(* IEC 61131-3 sources: Dev/Dev_V200/200 (part 18) *)

(* ---- _Nh_WEB.st ---- *)
(* KNIZNICA PRE FUNKCIE WEBMAKERU: HomePage,autologin, presmerovanie na volnu stranku a riadenie pristupu = usermanagement, *)

{ $ IFDEF __NH_WEB }

// hlavna obrazovka

// ************************** web ****************

FUNCTION _NhTchObjOK   {HIDDEN} : BOOL                                     // dotyk nad aktivnym objektom ( cm>0) na stranke
	VAR_INPUT
		///***26.6.24 skusmo pridane pre 109
		Qr			: BOOL;						// posle hned v 1.cykle po dotyku aj CMD, cim zabezpeci refresh a prijatie xA^.tch.Qr
		obj		: BOOL := true;
		cmd		: USINT;
	END_VAR
	IF Obj THEN
   	xA^.tch.cm     := xO^.cm;
	ELSE
		xA^.tch.cm     := cmd;
	END_IF;

   xA^.tch.row    := j;                               // tu sa vyplni ak by nebol browser
   xA^.tch.obj    := INT_TO_SINT(ix);
   xA^.tch.Q      := true;                            // centralny priznak, ze na nejakom objekte bol dotyk
   xA^.tch.Qr     := true;
   xO^.tch        := true;                            // priznak dotyku priamo na objekte, nuluje ho xA^.tch.Qf a do objektu uz nedojde
	xA^.tch.aObj	:= PTR_TO_UDINT( ADR(xO^) );
 	xO^.Q				:= true;									// nastavi sa Qr, zostane v objekte aj po Qf, objekt si ho spolu s Qf musi vynulovat sam
	IF Qr	THEN
		xA^.tch.CMD    := xA^.tch.cm;							// refresh v tom cykle je este xA^.tch.Qr := true
   	xO^.Qr			:= true;                         // cita sa v objekte, nuluje sa v dalsom cykle
	END_IF;
   ix             := 0;                                              // vykona sa exit s WHILE
   j              := 0;
   _NhTchObjOK       := true;

 	_Nh_Log_Evn_ADD(tsk := 200);

END_FUNCTION

FUNCTION _NhObjXY {HIDDEN}: BOOL                                     // dotyk nad aktivnym objektom ( cm>0) na stranke
   _NhObjXY := false;
   IF xA^.tch.x1 > xO^.x - x  AND
      xA^.tch.x1 < xO^.x + x  AND
      xA^.tch.y1 > xO^.y - y  AND
      xA^.tch.y1 < xO^.y + y  THEN

      _NhTchObjOK();
      _NhObjXY       := true;
   END_IF;
END_FUNCTION

FUNCTION _NhTchObj  {HIDDEN} : BOOL            // zaciatok noveho dotyky = hlada sa objekt
   VAR_TEMP
		wh2r		: BOOL;
      o        : INT;
      wh       : USINT;
//      whOld    : USINT;
	END_VAR
   _NhTchObj      := false;
   j  := USINT_TO_SINT(xM^.ixb[0].row.rws);
   WHILE _NhTchObj = false AND j > 0 AND xA^.tch.row < 0 DO
      IF xB^.r[ j ].h.nd > 0  THEN                                	// j = riadok
         xR    := ADR(xB^.r[ j ]);
         ix  	:= SINT_TO_INT(_RowObr);                              // ix = objekt; max.pocet objektov
         WHILE _NhTchObj = false AND  ix >= 0 DO                     // posupuje sa od posledneho objektu (je navrchu ) az k 0-temu, ktory je naspodku (oramovanie browsu)
				wh2r 	:=	false;
				IF ix > 0 THEN
            	xO    :=  ADR(xR^.o.ob[ix-1]);                           // predchadzajuci riadok
      			wh2r 	:= xO^.wh=123 OR  xO^.wh=109;							// preskoci aktualny riadok
				END_IF;
   			xO    :=  ADR(xR^.o.ob[ix]);
            IF wh2r 	 THEN
					;
            ELSIF xO^.nTch OR xO^.wh =  0 THEN
					;
            ELSIF xO^.wh = 13 THEN
            	o        		:= xO^.fn;
             	xS       		:= ADR(xB^.s[o]);
					IF xB^.s[xO^.fn].zom AND
						_NhTchObjXYW(	x	:=	xO^.x + xO^.w - 100,
											y 	:= xO^.y-50,
											w 	:= 100,
											h	:= 30 		 )	THEN

						xB^.s[xO^.fn].tun := NOT xB^.s[xO^.fn].tun;        // zmeni tun/sld/tun...
                  _NhTchObj      := _NhTchObjOK();
                  xO^.tch   		:= false;                                           // nastavi sa okamzite dotyk
                  xA^.tch.cmd    := xA^.tch.cm;                                           // nastavi sa okamzite dotyk
						xA^.tch.end		:= true;

         		ELSIF _NhTchObjXYW(	x	:=	xO^.x-15,
												y 	:= xO^.y-10,
												w 	:= xO^.w+30,
												h	:= 20 		 ) THEN

							IF (  xS^.bal AND xA^.tch.x1 > xS^.xv - 15 AND xA^.tch.x1 < xS^.xv + 15 ) // je zobrazena gulicka, dotyk na nej okamzite vyvola slider
                              OR
                           (  xA^.tch.x1 > xO^.x - 15 AND xA^.tch.x1 < xO^.x + 15)                // alebo dotyk okolo zaciatku
                              OR
                              xL^.brw = false   THEN

	                        _NhTchObj      := _NhTchObjOK();
  	                        xA^.tch.cmd    := xA^.tch.cm;                                           // nastavi sa okamzite dotyk
									xA^.tch.evn 	:= 6;

                     END_IF;
					END_IF;

            ELSIF xO^.wh = 14 THEN      // point-time SLIDER
            	IF xA^.tch.y1 > xO^.y - xO^.h AND                        // pod vrchom
                        xA^.tch.y1 < xO^.y + 50   AND                         // pod spodkom = obrazok
                        xA^.tch.x1 > xO^.x - 60    AND                        // pred zaciatkom
                        xA^.tch.x1 < xO^.x + xO^.w + 60    THEN               // za koncom
                        _NhTchObj      := _NhTchObjOK();

								xA^.tch.evn 	:= 6;
                        xA^.tch.cmd    := xA^.tch.cm;

						END_IF;

            ELSIF xO^.wh = 123 THEN      // vyber z volieb {riadkov} pod sebou  - NOVA VERZIA
               // tento objekt je dvojriadkovy, v druhom riadku sa vyhodnocuje WhOld z predch.riadka
               xOh := xO;
               IF xA^.tch.x1 >= xOh^.cf.x - 10                             AND     // 1.riadok zaciatok
                  xA^.tch.x1 <= xOh^.cf.x + xOh^.cf.w                         AND     // 1.riadok koniec
                  xA^.tch.y1 >= xOh^.cf.y - 20                             AND     // 1.riadok zaciatok
                  xA^.tch.y1 <= xOh^.cf.y + USINT_TO_INT(xOh^.cf.rw2)*xOh^.cf.h  THEN    // posledny riadok  (+10 je akokeby riadok naviac)

						_NhTchObj      := _NhTchObjOK(obj:=false,cmd:=205);
//                  xA^.tch.cm     := 251;
//                  xA^.tch.cm     := 205;
                  xOh^.tch       := true;                                           // priznak dotyku priamo na objekte

               END_IF;
//            ELSIF WhOld = 123 THEN       // prepinac medzi riadkami - NOVA VERZIA
               ;
            ELSIF xO^.wh = 103 THEN      // vyber z volieb {riadkov} pod sebou  - NOVA VERZIA
               ;
            ELSIF xO^.wh = 107 THEN      //  doplnujuce statusy na objektom
               IF _Nh_Web_SHW_107(tch:=true) THEN
                  _NhTchObj      := true;
               END_IF;
            ELSIF xO^.wh = 109 THEN      //  ROL * slider
            	xRo				:= xO;
               IF _NhxPt(c := xRo^.cf.c, n := xRo^.cf.n,x:=109) = false THEN
               	RETURN;
					END_IF;
               xRol 				:= xPt;
					xRol^.me.CMDs	:= 0;																		// reset
(*
					IF _NhxCfg(c := xRo^.cf.c, n := xRo^.cf.n, par := true, p := xRo^.cf.p, x:=20) = false THEN
						RETURN;
					END_IF;
*)

					del := USINT_TO_INT(xRo^.wObr);											// len prevod na INT - koli strukture

					IF xRo^.StatRow AND
						_NhTchObjXYW(		x := xRo^.xObrL - del/2 ,        				// dotyk nad ikonou LAM v stavovom riadku
												y := xRo^.yObr  - del/2 ,
												w := del,
												h := del) THEN
							_NhTchObj      := _NhTchObjOK( Qr:=true );
							xRol^.me.CMDs	:= 28;													// Lamely do opacneho smeru

					ELSIF xRo^.StatRow AND
							_NhTchObjXYW(	x := xRo^.xObrR - del/2 ,        				// dotyk nad ikonou ROL v stavovom riadku
												y := xRo^.yObr  - del/2 ,
												w := del,
												h := del) THEN
							_NhTchObj      := _NhTchObjOK( Qr:=true );
							xRol^.me.CMDs	:= 11;													// ROLETA prepnut

//					ELSIF xRol^.cx.etHandBlkWind > 0 AND														// bezi delay rucneho zasahu
					ELSIF xRol^.cx.CmdWind = 20 AND														// bezi delay rucneho zasahu
							_NhTchObjXYW(	x := xRo^.x + xRo^.w - xRo^.wObrInfo/2,		// zrusit delay rucneho zasahu
												y := xRo^.y - xRo^.wObrInfo/2,
												w := xRo^.wObrInfo,
												h := xRo^.wObrInfo) THEN
							_NhTchObj      := _NhTchObjOK( Qr:=true );
							xRol^.me.CMDs	:= 200;													// zrusit blokovanie

					ELSIF xRol^.cx.CmdWind = 10 AND												// bezi ochrana pred vetrom - restartnut
							_NhTchObjXYW(	x := xRo^.x - xRo^.wObrInfo/2,
												y := xRo^.y - xRo^.wObrInfo/2,
												w := xRo^.wObrInfo,
												h := xRo^.wObrInfo) THEN
							_NhTchObj      := _NhTchObjOK( Qr:=true );
							xRol^.me.CMDs	:= 201;													// restart WindGuard

					ELSIF xRo^.SldLam AND xRo^.tchLam AND										// slider LAM
							_NhTchObjXYW(	x := xRo^.xLam - 10 ,
												y := xRo^.yLam - xRo^.rCirSld/2,
												w := 20,
												h := xRo^.hLam + xRo^.rCirSld) THEN
							_NhTchObj      := _NhTchObjOK( Qr:=true );
							xA^.tch.evn 	:= 6;
							xRol^.me.CMDs	:= 72;													// slider LAM

    				ELSIF _NhTchObjXYW(	x := xRo^.x  ,											// plocha rolety aj s boxom nad
												y := xRo^.y - xRo^.bRol,
												w := xRo^.w ,
												h := xRo^.h + xRo^.bRol + xRo^.rCirSld ) THEN

							_NhTchObj      := _NhTchObjOK( Qr:=true );
							IF xRo^.SldRol THEN                                         // povoleny slider
								xA^.tch.evn 	:= 6;
								xRol^.me.CMDs	:= 71;												  	// slider ROL
							ELSIF xRo^.tchUpDn  THEN                             			// povolit prepnutie
								xRol^.me.CMDs	:= 1;														// prepni
							ELSE
								xRol^.me.CMDs	:= 3;														// stop
							END_IF;
					END_IF;
					IF _NhTchObj AND xRo^.chk = false AND xRol^.cx.CMD > 200 THEN
						xA^.tch.evn 	:= 0;
						xRol^.me.CMDs	:= 3;													// restart WindGuard
      			END_IF

            ELSIF xO^.wh = 22 OR xO^.wh = 121 THEN      														//  HET/VEN : AUTO-MAN/0/1/2/3
//					IF _NhTchObjXYW(x:=xO^.x-xO^.w/2, y:=xO^.y-xO^.w/2, w:=xO^.h * 4 + xO^.w, h := xO^.w) THEN
					IF _NhTchObjXYW(x:=xO^.x-xO^.w/2, y:=xO^.y-xO^.w/2, w:=xO^.h * USINT_TO_INT(xO^.cf.c) + xO^.w, h := xO^.w) THEN
						_NhTchObj      := _NhTchObjOK();
					END_IF;

            ELSIF xO^.wh = 21  THEN
					IF _NhTchObjXYW(x:=xO^.x-xO^.w/2, y:=xO^.y-xO^.w/2, w:=xO^.w, h := xO^.w) THEN
						_NhTchObj      := _NhTchObjOK();
					END_IF;

            ELSIF xO^.wh > 0 AND xO^.nTch = false THEN

               x     := xO^.w / 2 + 9;
               y     := x;             //***

               // xO^.h : 1 - obrazok s  podfarbenim
               // 6 - vypis textu :vyska
               // 10 - obrazok WSB
               // 13 - slider
               // 16 - bool premenna
               // 17 - akcie na obrazovke k WSB
               // 19 - vypisanie hodnoty premennej : style
               // 20 - chceck nad polom obrazkov
               // 21 - vypis textu s hodnotou
               // 90 - dash h=vyska       OK
               CASE xO^.wh OF
//                 22 :   wh := 20;
                120 :   wh := 255;
               ELSE     wh := xO^.wh;
               END_CASE;

               CASE wh OF
                  0 : ;                                              // prazdny objekt
                255 :   // objekt je urceny sirkou a vyskou, vo vnutri moze mat podobejky, ktore sa identifikuju v _Nh_SHW
                        IF xA^.tch.x1 >= xO^.x - xO^.h/2          AND      // spodna hranica = zaciatok - vyska/2
                           xA^.tch.x1 <= xO^.x + xO^.w + xO^.h    AND      // horna hranica
                           xA^.tch.y1 >= xO^.y - xO^.h/2          AND      // vrch
                           xA^.tch.y1 <= xO^.y + xO^.h/2  THEN             // spodok
                           _NhTchObj := _NhTchObjOK();
                        END_IF;

                  6 :   // click nad textom formatovany je zlava do prava
                     ok := xA^.tch.y1 > xO^.y - 20 AND xA^.tch.y1 < xO^.y + 20;
                     CASE xO^.fn  OF
                       2 : // na stred
                           ok := ok AND xA^.tch.x1 > xO^.x - xO^.w/2 AND xA^.tch.x1 < xO^.x + xO^.w/2;
                       1 : // z prava do lava
                           ok := ok AND xA^.tch.x1 > xO^.x - xO^.w AND xA^.tch.x1 < xO^.x;

                     ELSE  // zlaba do prava
                           ok := ok AND xA^.tch.x1 > xO^.x AND xA^.tch.x1 < xO^.x + xO^.w;

(*
                        IF xA^.tch.x1 > xO^.x           AND
                           xA^.tch.x1 < xO^.x + xO^.w   AND
                           xA^.tch.y1 > xO^.y - 20   AND
                           xA^.tch.y1 < xO^.y + 20 THEN
                           _NhTchObj      := _NhTchObjOK();
                        END_IF;
*)
                     END_CASE;
                     If ok THEN
                        _NhTchObj      := _NhTchObjOK();
                     END_If;

                 15 : // typovy DAY + PO-NE
                        xPtD  := ADR(xO^.cf.n);                                                             // na adrese xO^.cf.n + xO^.cf.p je adresa premennej v UDINT
                        xPoD  := UDINT_TO_PTR(xPtD^);

                        _Nh_FRM_Read(frm:=248);   // sablona PO-NE pre DAY,HET,VEN
                                                                       // pointer riadiacej jstruktury dna
                        xM^.pod.po.Btn := false;
                        IF    xA^.tch.y1 > xO^.y - 40 AND                                    // vrchny okraj typovyc dni
                              xA^.tch.y1 < xO^.y + 85+35 THEN                                // spodny okraj PO-NE
                           // sme v objekte
                           FOR i := 0 TO 11 DO
                              IF i > 0 AND i < 8 THEN
                                 y := xO^.y + 85;                                         // dni Pon-Ned
                              ELSE
                                 y := xO^.y;
                              END_IF;
                              IF xA^.tch.y1 < y + 40 AND                                  // nad spodkom
                                 xA^.tch.y1 > y - 40 AND                                  // pod vrchom
//                                 xA^.tch.x1 < xO^.x + _ObjDay.xDay[i]+40 THEN             // pred koncom objektu
                                 xA^.tch.x1 < xO^.x + yFrm_248.xDay[i]+40 THEN             // pred koncom objektu

                                 xM^.pod.po.Btn := xM^.pod.po.Day = i;                            // stlaceny ten isty BTN
                                 IF xM^.pod.cp.cpy THEN                                       // je oznacene kopirovanie
                                    IF xM^.pod.po.Btn = false THEN                            // vymazat vsetko ku kopirovaniu
                                       xM^.pod.cp.dst[i] := NOT xM^.pod.cp.dst[i];
                                    END_IF;
                                 ELSIF i = 0 THEN                                         // prepli sme na hlavmu ikonu prac.dni
                                    IF xPoD^.Day=0 OR xPoD^.Day > 7 THEN                  // predtym bola ina hlavna ikona
                                       xPoD^.Day := _Nh_Poi_Home_Day();                        // nastavi sa aktualny day
                                    END_IF;
                                    xM^.pod.po.Day := xPoD^.Day;
                                 ELSE

                                    IF xPoD^.Day = 0 THEN
                                       xPoD^.Day := i;                                    // prepnutie na iny den a ked je fix prepise Day
                                    END_IF;
                                    xM^.pod.po.Day := i;
                                 END_IF;
                                 _NhTchObj   := _NhTchObjOK();
                                 EXIT;
                              END_IF;
                           END_FOR;
                        END_IF;

                 10 : // akcie od WSB, typ spotrebica (v xO^.h je cislo obrazka)
                     _NhTchObj   := _NhObjXY();

                 17 : // akcie od WSB, typ spotrebica (v xO^.h je cislo obrazka)
                     _NhTchObj   := _NhObjXY();
                 19 : // text
(*
                  GTEXT_STYLE_ITALIC + GTEXT_STYLE_ALIGN_LEFT   + GTEXT_STYLE_HRIGHT  + GTEXT_STYLE_VCENTER,    // stred riadka zlava do prava
                  GTEXT_STYLE_ITALIC + GTEXT_STYLE_ALIGN_RIGHT  + GTEXT_STYLE_HLEFT   + GTEXT_STYLE_VCENTER,    // stred riadka, zprava do lava
                  GTEXT_STYLE_ITALIC + GTEXT_STYLE_ALIGN_CENTER + GTEXT_STYLE_HCENTER + GTEXT_STYLE_VCENTER,    // stred riadka, stred textu
                  GTEXT_STYLE_NORMAL + GTEXT_STYLE_ALIGN_LEFT   + GTEXT_STYLE_HRIGHT  + GTEXT_STYLE_VDOWN,       // zhora-dolu, zlava do prava
                  GTEXT_STYLE_NORMAL + GTEXT_STYLE_ALIGN_RIGHT  + GTEXT_STYLE_HRIGHT  + GTEXT_STYLE_VDOWN       // zhora-dolu, zlava do prava
*)
                     IF xO^.fn = 0 THEN
//                        y := xO^.h/2+5;
                        y := xO^.h*2  ;
                        CASE xO^.BgC OF
                          0 : x := -xO^.w/2;
                          1 : x := xO^.w/2;
                          3 : ;
                          4 : ;
                        END_CASE;
                        IF xA^.tch.y1 > xO^.y - y AND                        // pod vrchom
                           xA^.tch.y1 < xO^.y + y   AND                         // pod spodkom = obrazok
                           xA^.tch.x1+x > xO^.x - xO^.w/2    AND                        // pred zaciatkom
                           xA^.tch.x1+x < xO^.x + xO^.w/2    THEN               // za koncom
                           _NhTchObj      := _NhTchObjOK();
                        END_IF;
                     ELSE
                        _NhTchObj := _NhObjXY();
                     END_IF;

                 27 : // viac BOOL premennych v poli za sebou (DayMode+LOCK)
                        IF _NhObjXY() THEN
                           xO^.tch := 1;
                           _NhTchObj := true;
                        END_IF;

                 20 : // viac BOOL premennych v poli za sebou (DayMode+LOCK)
                     IF xO^.cf.c > 0 AND xO^.h = 0 THEN  // viac objektov na sebe, cislo objektu je ulozene v premennej, ktora je USINT, prepne na dalsi objekt
                        IF _NhObjXY() THEN
                           _NhTchObj := true;
                           xPtD  := ADR(xO^.cf.n);                                                             // na adrese xO^.cf.n + xO^.cf.p je adresa premennej v UDINT
                           xPtU  := UDINT_TO_PTR(xPtD^);
                           IF xPtU^ < xO^.cf.c THEN
                              xPtU^ := xPtU^ + 1;
                           ELSE
                              xPtU^ := 0;
                           END_IF;
                        END_IF;
                     ELSE
                        x := xO^.w/5*3;
                        IF xA^.tch.x1 > xO^.x - x  AND                            // tesne pred prvym obrazkom
                           xA^.tch.x1 < xO^.x + x + xO^.h * USINT_TO_INT(xO^.cf.c)  AND       // tesne za poslednym obrazkom
                           xA^.tch.y1 > xO^.y - x  AND
                           xA^.tch.y1 < xO^.y + x  THEN
                           _NhTchObj      := _NhTchObjOK();
                        END_IF;
                     END_IF;

                 23 :   // prepinac viac riadkov pod sebou
                        y := USINT_TO_INT(xO^.cf.c);
                        IF xA^.tch.x1 > xO^.x - 10          AND     // zaciatok komponenty
                           xA^.tch.x1 < xO^.x + xO^.w + 10  AND     // koniec
                           xA^.tch.y1 > xO^.y - 20          AND     // 1.riadok
                           xA^.tch.y1 < xO^.y + (xO^.fn * y) + 20   // posledny riadok
                                 THEN
                           _NhTchObj   := _NhTchObjOK();
                           o           := xO^.y + xO^.fn/2;
                           FOR i := 1  TO xO^.cf.c DO
                              IF xA^.tch.y1 < o THEN
                                 xFmt23      := ADR(xO^.fmt);
                                 xFmt23^.obj := i;
//                                 xA^.tch.prs := false;
                                 EXIT;
                              END_IF;
                              o := o + xO^.fn;
                           END_FOR;
                        END_IF;

//                 21 :   // prepinac viac riadkov pod sebou
//   	                  y     := x;
//	   	               _NhTchObj := _NhObjXY();

               ELSE
                  IF xO^.h <= 0 THEN
                     y     := x;
                  ELSE
                     y     := xO^.h / 2 + 9;
                  END_IF;
                  _NhTchObj := _NhObjXY();
               END_CASE;
            END_IF;
            IF _NhTchObj THEN
               RETURN;
            END_IF;
            ix       := ix - 1;
//            ix       := ix + 1;
//            WhOld    := xO^.wh;                 // pre dvojriadkove objekty (123..)

         END_WHILE;
      END_IF;
      j := j - 1;
   END_WHILE;
END_FUNCTION

FUNCTION _NhTchMnu {HIDDEN} : BOOL      // najde riadok a v nom objekt na ktorom bol dotyk
  _NhTchMnu       := false;

  xA^.tch  := _eTch;
  aWht     := _eWht;

   xA^.tch.x1     := xCan^.touch.x;
   xA^.tch.x2     := xCan^.touch.x ;
   xA^.tch.y1     := xCan^.touch.y;
   xA^.tch.y2     := xCan^.touch.y;

   jj    := 8;                                                 // prechadzaju sa vsetky menu
   rb    := false;
   IF xM^.edt  THEN
      jj := 1;                                                                // testuje sa len CANCEL
   ELSIF xB^.rw > 0 AND xL^.brw THEN                                          // ak je browser a su naplnene nejake riadny, najskor pg navigator
      IF _NhTchXY(v := xA^.tch.y1, v1 := ky2, v2 := ky2, xy:= 30 ) THEN         // dotyk okolo  spodnej ciary
         x := xIxB^.x1;
         FOR i := 1  TO xIxB^.n DO
            IF _NhTchXY(v := xA^.tch.x1, v1 := x, v2 := x, xy := 30 ) THEN     // dotyk nad bodom
               IF xIxB^.idx > xIxB^.row.rws THEN                               // mame viac dat zaznamov ako je riadkov
                  IF i = xIxB^.n THEN                                          // posledny index
                     i := xIxB^.idx - xIxB^.row.rws + 1;
                  ELSIF i = 1 THEN                                             // 1.index
                     ;
                  ELSE
                     i := (i-1) * xIxB^.row.rws  + 1;                          // vypocita sa
                  END_IF;
               ELSE
                  i := 1;
               END_IF;
               _Nh_Map_Idx(ixb := 0, idx := i);                                  // namapuje najdeny index
               xIxB^.ix1   := i;                                               // toto asi nemusi byt
               xL^.rw1     := xIdx^.ix[aWeb.nbr].dev;                              // do 1.riadku sa vlozia data
               xA^.tch.cmd := 252;                                             // vypis a predefinovanie dat od noveho 1-veho riadka
               _NhTchMnu   := true;
               RETURN;
            END_IF;
            x := x + USINT_TO_INT(xIxB^.w);
         END_FOR;

			// dotyk na spodnej ciare mimo PG-navigator tu sa meni mierka yk:=1.0 .... yk       := MIN(xUsr^.cx.IP[1].y, 1.14) ;

		END_IF;
      ;
   END_IF;
   FOR j := 1  TO jj DO
      xOm  := ADR(xU^.o[j]);
      IF xOm^.fn > 0 AND  xOm^.cm > 0 AND
         _NhTchXY(v := xA^.tch.x1, v1 := xOm^.x, v2 := xOm^.x, xy:= xOm^.w/7*4 )  AND // sirka
         _NhTchXY(v := xA^.tch.y1, v1 := xOm^.y, v2 := xOm^.y, xy:= xOm^.w/7*4 )    // vyska
            THEN
         xA^.tch.obj  := j;
         xA^.tch.cm   := xOm^.cm;
         IF xL^.obj = 200 AND xA^.tch.obj > 2 THEN              // stlacene spodne menu v SETUP
            xA^.tch.cmd    := 200;
         ELSE
            xA^.tch.cmd  := xA^.tch.cm;
         END_IF;
         _NhTchMnu    := true;
         EXIT;
      END_IF;
   END_FOR;
   IF xM^.edt  THEN                                            // edituje sa nazov
      IF _NhTchMnu THEN
         xM^.new := -1;
      END_IF;
       xA^.tch.cmd      := 100;                                // aktivuje CMD editaciu okamzite
      _NhTchMnu         := true;
   ELSIF xA^.tch.x1 > xc - 150         AND                     // dotyk na nazve
         xA^.tch.x1 < xc + 150         AND
         xA^.tch.y1 > xU^.o[1].y - 20  AND                     // vyska nazvu
         xA^.tch.y1 < xU^.o[1].y + 20 THEN

      IF xF^.cf.c = 0 OR xF^.cf.n = 0 THEN                     // nazvy su z aLang
            ;
      ELSIF xM^.set THEN
         rb := aCfg[xL^.fil.cf.c].edn;                         // cfg, vratane nazvy Moj domov co je acfg[3] = zone
      END_IF;
      IF rb THEN
//			xA^.trg.Qr     := 0;
//			xA^.trg.Qf     := 0;
//			xA^.trg.Q      := 0;
         xA^.tch.cmd    := 101;                                // aktivuje CMD editaciu okamzite
         xM^.edt        := true;                               // pri modifikacii nazvu sa to oznaci hned
         _NhTchMnu      := true;
      END_IF;
   END_IF;
END_FUNCTION

FUNCTION_BLOCK _NhWebAcces   {HIDDEN}
   VAR_TEMP
      s        : USINT;
      sa       : USINT;
//      new      : STRING[14];
   END_VAR
   GetWebServerAccess(accessTable := aAcc.wA);
   IF aAcc.wA <> aAcc.wO OR SYSTEM_S.F_EDGE_1SEC THEN
      aAcc.WebChg := aAcc.WebChg + 1;                                         // pocet zmien
      memset(0, sizeof(aAcc.pgN), void(aAcc.pgN));                          // vymazat novy pg, ktorasa bude naplnat
      ii := aWeb.A[1].usr;
      FOR aWeb.nbr := 1 TO _Nh_WEB_M DO
         aWeb.A[ aWeb.nbr ].usr := 0;
      END_FOR;
      FOR s := 0 TO 7 DO
         sa    := _webState(s := aAcc.wA[s].state);
         IF sa = 3  THEN                                                      // zaujima nas len stav 3
            yTx3  := MID(aAcc.wA[s].lastFile,8,5);                            // "/002_NHM.XML" .... '_NHM.XML'
            IF yTx3 = '_NHM.XML' THEN                                           // nova stranka je Mx                           OK
               yTx3  := MID(aAcc.wA[s].lastFile,3,2);
               i := STRING_TO_USINT(yTx3);
               IF i <= _Nh_WEB_M THEN
                  aWeb.A[ i ].usr := i;
                  IF aWeb.M[ i ].naz = '' AND  aWeb.M[ i ].new < 1 THEN
                     aWeb.A[ i ].tch.cmd := 20;                   // vytvori sa nova obrazovka
                     aWeb.M[ i ].lvl     := 0;
                  END_IF;
               END_IF;
            END_IF;
         END_IF;
      END_FOR;
      IF aWeb.A[1].usr > 0 AND ii > 0 THEN
//         aWeb.A[1].usr := ii;
      END_IF;
      aAcc.wO  := aAcc.wA;                                            // vyrovna data
   END_IF;
END_FUNCTION_BLOCK

FUNCTION_BLOCK _NhWebControl    {HIDDEN}
  	VAR
      fbNhWebAcces : _NhWebAcces;
  	END_VAR
      fbNhWebAcces();                                                // riadenie pristupu na webserver
      // prechadza nadefinovane stranky
      FOR aWeb.nbr := 1 TO _Nh_WEB_M DO
//         IF aAcc.pgN.pg[aWeb.nbr].usage > 0 THEN                   // aktivna stranka
         xA       := ADR( aWeb.A[ aWeb.nbr ] );                      // dotk,canvas..
         IF xA^.usr > 0 THEN                                         // aktivna stranka
            xM       := ADR( aWeb.M[ aWeb.nbr ] );                   // zakladne data stranky
            xB       := ADR( xM^.brw );                              // browser
            xU       := ADR( xM^.mnu[ aWeb.M[aWeb.nbr].lvl ]);                            // menu
            xL       := ADR( xM^.lvd[ aWeb.M[aWeb.nbr].lvl ]);                            // data k browsu
            xCan     := ADR( aWeb.A[ aWeb.nbr ].can );               // canvas
            xA^.trg(In := xCan^.touch.y > -32767 );                  // zistenie dotyku
            _NhxUsr(u := xA^.usr );                                  // pri vstupe do session namapuje usra, potom uz v programe nikdy
            xA^.admin   := aWeb.nbr = 1;
            IF xUsr^.cx.sbj = 0 OR xUsr^.cx.sbj > INT_TO_USINT(aCfg[3].rec) THEN
               xA^.sbj     := 1;
            ELSE
               xA^.sbj     := xUsr^.cx.sbj;
            END_IF;
            xA^.admin      := aWeb.nbr    = 1;
            IF xA^.admin THEN
               xA^.UsrRight   := 9;
            ELSE
               xA^.UsrRight   := xUsr^.cx.UsrRight;
            END_IF;
            IF xUsr^.cx.IP[1].y > 1.0 THEN
               yk       := MIN(xUsr^.cx.IP[1].y, 1.14) ;
               yk       := MIN(xUsr^.cx.IP[1].y, 1.5) ;
            ELSE
               yk       := 1.0;
            END_IF;
            ky2      := REAL_TO_INT( INT_TO_REAL(yy2)*yk);
            IF xUsr^.cx.IP[1].y <> xUsr^.cx.IP[2].y THEN                                     // zmena vysky zobrazenia
               xA^.hom           := true;                                                    // vytvori sa nova obrazovka
               xUsr^.cx.IP[2].y  :=  xUsr^.cx.IP[1].y;
            END_IF;

            // VYHODNOTENIE DOTYKU - PRIRADENIE AKCIE
            // 1 - potiahnutie dolu
            // 2 - potiahnutie hore
            // 3 - potiahnutie dolava
            // 4 - potiahnutie doprava
            // 5 - dotyk
            // 6 - PRESS

				xA^.tch.Qr	:= false;
				xA^.tch.Qf	:= false;
            IF xA^.hom THEN
               xM^.naz     := '';
               xA^.tch.cmd := 20;                                                // prekresli sa nova obrazovka
               xM^.lvl     := 0;
               xA^.hom     := false;
   			ELSIF xA^.trg.Qr THEN                                                // prvy dotyk zisti ci bol na nejakom objekte
               IF _NhTchMnu() THEN                                               // najskor skusi menu
                  xA^.tch.End := true;                                           // natvrdo ukoncit , necaka sa za Qf
                  xA^.tch.Mnu := true;                                           // natvrdo ukoncit , necaka sa za Qf
                  xA^.tch.evn := 1;                                              // kod dotyku
                  xM^.htt     := '';                                             // zrusi pripadnu externu stranku
               ELSIF _NhTchObj() THEN
(*
                  IF xA^.tch.cmd > 0 THEN                                        // prisiel fixny EVN, vzdy ma prednost
                     ;
                  ELSIF xL^.brw = false AND xO^.prs = false THEN                  // NIE-je browser, ALEBO objekt nema povoleny pres
                     xA^.tch.evn := 5;
                     xA^.tch.cmd := xA^.tch.cm;
                  END_IF;
*)
               ELSE                                                              // dotyk mimo objektu
                  xA^.tch.cm  := 254;                                            // kompletny refresh od 1. riadku
						xA^.tch.End	:= 1;
               END_IF;

				ELSIF xA^.trg.Qf THEN                                                // koniec dotyku alebo press
					xA^.tch.Qf		:= 1;
					xA^.tch.End    := 1;
					IF xA^.tch.aObj > 0 THEN
						xO					:= UDINT_TO_PTR(xA^.tch.aObj);
						xO^.Qf			:= true;
						IF xA^.tch.evn = 6 THEN
     						xA^.tch.cmd := xA^.tch.cm;
						ELSIF xA^.tch.evn = 0 THEN
///***							xA^.tch.evn := 4;
     						xA^.tch.cmd := xA^.tch.cm;
						END_IF
      			END_IF;

				ELSIF xA^.tch.cmd > 0 THEN                                           // nieco nasilne obieha dookola (rolovanie)
					IF xA^.tch.aObj > 0 THEN
						xO					:= UDINT_TO_PTR(xA^.tch.aObj);
						xO^.Qr			:= false;
//						xO^.Dummy1		:= 1;
					END_IF;
					;
            ELSIF xA^.trg.Q THEN                                                   // fyzicky pokracuje dotyk
               xA^.tch.tme := xA^.tch.tme + aSys.mSec;
               xA^.tch.x2  := xCan^.touch.x ;                                       // suradnica po posunuti
               xA^.tch.y2  := xCan^.touch.y ;
					IF xA^.tch.aObj > 0 THEN
						xO					:= UDINT_TO_PTR(xA^.tch.aObj);
						xO^.Qr			:= false;
                  IF xL^.brw = false AND xO^.prs  THEN                  // NIE-je browser, ALEBO objekt nema povoleny pres
							IF xA^.tch.tme > 800 THEN
								xA^.tch.evn := 6;
							ELSE
								xA^.tch.evn := 5;
							END_IF;
						END_IF;
					END_IF;
               IF xA^.tch.End 	THEN                                 				// fyzicky je dotyk, ale uz je vyhodnoteny Up-Dn-Left-right
						xA^.tch.cmd := 0;
						///***28.6.24
						xO^.tch		:= false;
						IF xA^.tch.aObj > 0 THEN
							xO^.Q		:= false;
   					END_IF;
					ELSIF xA^.tch.evn = 0 THEN
                  IF xA^.tch.y2 - xA^.tch.y1 > 20 THEN                                 // dolu
                     xA^.tch.evn := 1;
//                     ok          := true;
                  ELSIF xA^.tch.y1 - xA^.tch.y2 > 20 THEN                              // hore
                     xA^.tch.evn := 2;
//                     ok          := true;
                  ELSIF xA^.tch.x1 - xA^.tch.x2 > 100 THEN                              // potiahnutie dolava
                     xA^.tch.evn := 3;
//                     ok2         := true;
                  ELSIF xA^.tch.x2 - xA^.tch.x1 > 100 THEN                              // potiahnutie doprava
                     xA^.tch.evn := 4;
//                     ok2         := true;
                  END_IF;
						IF xA^.tch.evn > 0 THEN
							xO^.tch		:= false;									////30.11.23 - pri rolovanisa zapinali objekty het/tve
///***							xA^.tch.obj	:= 0;
							xA^.tch.End := 1;
	     					xA^.tch.cmd := xA^.tch.evn;
						END_IF;
					ELSIF xA^.tch.evn = 6 THEN
     					xA^.tch.cmd := xA^.tch.cm;
					ELSIF xA^.tch.evn = 5 THEN
     					xA^.tch.cmd := xA^.tch.cm;
					END_IF;
				ELSIF xA^.tch.End THEN                                                // koniec dotyku alebo press
					IF xA^.tch.aObj > 0 THEN
						xO					:= UDINT_TO_PTR(xA^.tch.aObj);
						xO^.tch			:= false;
						xO^.Qf			:= false;
						xO^.Q				:= false;
						xA^.tch.aObj	:= 0;
      			END_IF;
					xA^.tch.End    := 0;
					xA^.tch.Q		:= 0;
					xA^.tch.cmd 	:= 0;
				END_IF;

            IF xA^.tch.cmd > 0 THEN                            // akcia od dotyku, nieco sa ma vykonat a v dalsom kole zobrazit
//               _Nh_Web_CMD(m := aWeb.M[aWeb.nbr]);             // zisti sa co sa ma vykonat
               aWeb.go     := true;                           // aby sa nevykonalo 2x
               aWeb.trg(rst := true, in := true);              // pripravi FB aby v dalsom cykle bol Qr
            ELSE                                               // ziadna akcia
               IF xL^.obj = 0 THEN                             // HOME
                  IF xHom^.ok.ref AND SYSTEM_S.R_EDGE_1SEC THEN
                     aWeb.trg.in := true;
                     aWeb.trg.Q  := false;                           // aby sa zabezpecil Qr
                     xHom^.ok.ref := false;                    // vynuluje sa poziadavka DEV
                  END_IF;
               ELSE
                  // zabezpecit refesh FRAME a HOME SCREEN
                  ok := SYSTEM_S.R_EDGE_1SEC;
                  IF ok THEN
                     IF xU^.o[8].fn > 50 THEN                           // zapnuty filter. Browser nemusi mat nic zobrazene
                        aWeb.trg.in := true;
                        aWeb.trg.Q  := false;
                     ELSE
                        FOR  i := 0  TO xB^.rw DO                       // hlada sa zobrazene DEV pre xM stranku
                           IF xB^.r[i].h.cf.c > 0  THEN
										IF xB^.r[i].h.cf.c = 2 THEN
											;
										ELSIF	_NhxPt(c := xB^.r[i].h.cf.c, n := xB^.r[i].h.cf.n,x:=49) THEN
											IF xPt^.ok.ref THEN                       // poziadavka DEV na refresh nastartuje refresh
   	                              aWeb.trg.in := true;
      	                           aWeb.trg.Q  := false;                           // aby sa zabezpecil Qr
         	                        xPt^.ok.ref := false;                  // vynuluje sa poziadavka DEV
            	                     ok          := false;
               	               END_IF;
										END_IF;
                           END_IF;
                        END_FOR;
                        IF ok AND xHom^.ok.ref THEN                     // nebol ziadny refresh, a v celom systeme bola zmena
                           IF xU^.o[8].fn > 50 THEN                     // zapnuty ON-filter
                              aWeb.trg.in := true;
                              aWeb.trg.Q  := false;
                           END_IF;
                        END_IF;
                     END_IF;
                  END_IF;
               END_IF;
               aWeb.trg();
               IF aWeb.trg.Qr THEN
///                  aWeb.trg.cm := 2;
                  aWeb.trg.et := 400;
                  aWeb.Go     := true;
               ELSIF aWeb.trg.Qe THEN
(*
                  IF aWeb.trg.cm > 0 THEN
                     aWeb.trg.cm := aWeb.trg.cm - 1;
                     aWeb.trg.et := 650;
                  ELSE
                      aWeb.trg.in := false;
                  END_IF;
*)
                  aWeb.Go     := true;
               END_IF;
               IF aWeb.Go  THEN
                  // vymysliet typ refreshu
                  IF xU^.o[8].fn > 50 THEN                                                // zapnuty ON-filter
                     xA^.tch.cmd := 254;                                                             // uplne novy vypis
                  ELSE
                     xA^.tch.cmd := 252;
                  END_IF;
               END_IF;
            END_IF;
            IF aWeb.Go THEN
               IF xA^.tch.row > 0 THEN
                  j  := xA^.tch.row;
                  xR := ADR(xB^.r[ j ]);
                  IF xR^.h.cf.c > 0 AND xR^.h.cf.c <> 2 THEN
                     _NhxPt(c := xR^.h.cf.c, n := xR^.h.cf.n,x:=50);
                     xDev := xPt;
                  END_IF;
               END_IF;

               _Nh_Web_CMD();

               aWeb.nrf := aWeb.nrf  + 1;
               aWeb.Go  := false;
            END_IF;
            xM^.frm  := xM^.htt <> '';                                                    // schova iFame = vnorena web stranka
         END_IF;
      END_FOR;

END_FUNCTION_BLOCK

(* ---- _Nh_Web_BRW.st ---- *)
{ $ IFDEF __NH_WEB }

FUNCTION _NhSetObjDsh   {HIDDEN}  : BOOL        // zobrazi Day a sumrk pre ROM,ZON,PIR
   VAR_INPUT
      grp      : USINT;
//      row      : USINT;
   END_VAR
   VAR_TEMP
      sld6     : BOOL := true;
   END_VAR
   _NhSetObjDsh := true;
   _NhxDev(c := xR^.h.cf.c, n := xR^.h.cf.n, x:=12 );
   CASE grp OF
		0 : ;
   ELSE	;

   END_CASE;
   If sld6 THEN
      IF xL^.dsh > 1 THEN                                            // posunut browser namiesto FAV
         xR^.o.ob[6].x     := xR^.o.ob[5].x ;
         xR^.o.ob[6].w     := 150 ;
         xR^.o.ob[5].x     := xR^.o.ob[3].x ;                        //
         xR^.o.ob[3].wh    := 0;                                     // FAV sa nevykonava
         xR^.o.ob[4].wh    := 0;                                     // FAV sa nevykonava
      END_IF;
      IF xL^.dsh = 3 THEN                                            // najmensi dash nema slider
//         xR^.o.ob[6].wh    := 0 ;
      END_IF;
   END_IF;

END_FUNCTION

FUNCTION _NhShwDay   {HIDDEN}  : BOOL                 // zobrazi Day a sumrk pre ROM,ZON,PIR
   VAR_INPUT
      rom   : BOOL := true;               // dalsi nastavenia pre ROM
//      day   : BOOL ;                      // zobrazi aj slniecko =den
      cf    : USINT := 1;
      nr    : USINT;

   END_VAR
   _NhShwDay := false;
   IF nr = 0 THEN                         // nepriradene cislo miestnosti
      xR^.o.ob[ 2].wh   :=  0;
//      xR^.ob[ 4].cm   := 22;
      xR^.o.ob[ 9].cm   := 6;
      xR^.o.ob[ 9].cf.c := 0;
      xR^.o.ob[ 9].cf.n := 359;
      xR^.o.ob[10].cf.c := 0;
      xR^.o.ob[10].cf.n := 358;

      RETURN;

   END_IF;

   _NhxPt(c := cf, n := USINT_TO_INT(nr),x:=44); xRom := xPt;
   // zobrazenie sumraku vlavo hore nad ikonou
(*
   IF xRom^.cx.Dark THEN
      _NhSetObjBrw(wh:=4, ob:=7, w := xR^.o.ob[7].w, h:= xR^.o.ob[7].w, o1 := USINT_TO_INT(_NhListObr.Dark[1]), c:=1 ,n:=1, cm := 200, vb := adr(vr)  );
   END_IF;
   // zobrazenie DayObr vpravo hore nad ikonou
   IF xRom^.cx.DayObr > 0 OR day THEN
      _NhSetObjBrw(wh:=4, ob:=8,  w := xR^.o.ob[8].w, h:= xR^.o.ob[8].w, o1 := USINT_TO_INT(_NhListObr.Day[1,xRom^.me.DayObr]), c:=1 ,n:=1, cm := 200, vb := adr(vr)  );
   END_IF;
*)
(*  ///???

   IF rom THEN
      IF  xL^.psn THEN                                         // nadefinuje zobrazenie LOCK btn
         ok := 0;
         IF xRoW^.stat > 4 THEN
            i := 7; ix := 94; z:= 80;                         // Alarm
         ELSIF xRoW^.Lock AND xRoW^.Full THEN
            i := 7; ix:= 69; z:= 72;
         ELSIF xRoW^.Lock THEN
            i := 6; ix:= 68; z:= 72;
         ELSE
            i := 0; ix:= 66; z:= 72;
         END_IF;
         _NhSetObjBrw(wh:=12, ob:=2, w:=z, h:=z+10, o1:=ix, FgC:=0, Bgc:=i , x:= xR^.o.ob[2].x, y:= xR^.o.ob[2].y , vb := adr(vr), cm:=28, btn:=ok);
         CASE xRoW^.stat OF
           0 : i := 0;
//           1 : i := 0;
           2 : i := 7; ix := 69;                               // zamyka sa - odchod
           3 : i := 8; ix := 89;                               // prichod, caka sa na kod
           4 : i := 7; ix := 291;                              // strazenie - pes
         ELSE
            IF xRoW^.MemAlarm THEN
               i := 7; ix := 94;                               // zapamatany alarm
            ELSE
               i := 0;
            END_IF;
         END_CASE;

         IF i > 0 THEN
            _NhSetObjBrw(wh:=12, ob:=6, w:=46, h:=56, o1:=ix, FgC:=1, Bgc:=i , x:= xR^.o.ob[2].x-xR^.o.ob[2].h/2, y:= xR^.o.ob[2].y-xR^.o.ob[2].h/5 , vb := adr(vr), nTch:=1, btn:=1 );
         END_IF;
      ELSE                                                     // nadefinuje zobrazenie teploty
         xR^.o.ob[2].cm   := 30;
//         xR^.o.ob[2].cm   := 30;

//         _NhSetObjBrw(ob:=2, wh:=219, w:=80, h := _Nh_O12(xL^.dsh<3,30,25), cm:=30, vb := adr(xDev^.al.ou.val), BgC:=1);
      END_IF;
*)

      xR^.o.ob[10].cm   := 30;                                 // dotyk nad nazvom = vnorit sa
      IF cf = 1 AND xL^.dsh =1 THEN
         xR^.o.ob[9].cf.c:= 254;
         xR^.o.ob[9].fmt := LEFT(xRom^.cf.ID,3);
         xR^.o.ob[9].fmt := insert(xRom^.cf.ID,'.',2) ;
      ELSE
         xR^.o.ob[9].wh    := 0;                                  // disable nazov 2
      END_IF;
      xR^.o.ob[5].wh    := 5;                                  // zobrazenie sumarov
      CASE xL^.dsh OF
           3 : // 12*2
               xR^.o.ob[5].y   := xR^.o.ob[5].y-30;
               xR^.o.ob[5].x   := xR^.o.ob[5].x-10;
               xR^.o.ob[5].w   := 35;
               xR^.o.ob[5].h   := 33;

               xR^.o.ob[2].y   := xR^.o.ob[3].y+5;               // presunie teplotu u ROM dolu, aby bolo vidiet naov room

               IF rom = false THEN
                  xR^.o.ob[2].w   := xR^.o.ob[2].w-10;
                  xR^.o.ob[2].h   := xR^.o.ob[2].h-10;
                  xR^.o.ob[2].fn  := 0;                        // aby  sa zobrazil stav DEV, inak je to naformatovanie hodnoty zprava do lava
               END_IF;
           2 :
               xR^.o.ob[5].y   := xR^.o.ob[5].y-45;
               xR^.o.ob[5].x   := xR^.o.ob[5].x-48;
               xR^.o.ob[5].w   := 35;
               xR^.o.ob[5].h   := 33;
               xR^.o.ob[2].w   := xR^.o.ob[2].w+xR^.o.ob[2].w/4;
               xR^.o.ob[2].h   := xR^.o.ob[2].h+xR^.o.ob[2].h/4;
         ELSE
               xR^.o.ob[5].y  := xR^.o.ob[5].y - 5;
      END_CASE;
(* ///???
      IF xRoW^.Body  THEN                                      // pohyb v rom/zone
         xR^.o.ob[0].FgC  := 3;
         xR^.o.ob[0].BgC  := 1;
      ELSIF xRoW^.stat > 4 THEN                                // narusenie
         xR^.o.ob[0].FgC  := 1;
//         xR^.o.ob[0].BgC  := 28;
         xR^.o.ob[0].BgC  := 7;
      ELSIF xRoW^.Lock AND xRoW^.Full THEN                     // uplne zamknutie
         xR^.o.ob[10].FgC  := 4;
         xR^.o.ob[0].FgC  := 1;
//         xR^.o.ob[0].BgC  := 7;
         xR^.o.ob[0].BgC  := 6;
      ELSIF xRoW^.Lock THEN                                    // ciastocne zamknutie
         xR^.o.ob[10].FgC  := 4;
         xR^.o.ob[0].FgC  := 1;
         xR^.o.ob[0].BgC  := 16;

      END_IF;
   END_IF;
*)

   _NhShwDay := true;
END_FUNCTION

FUNCTION _NhRowDSH {HIDDEN} : BOOL           //   NAPLNI RIADOK FIXNYMI HODNOTAMI
   VAR_INPUT
      row      : USINT;
   END_VAR
   _NhRowDSH  := true;

//   yTx3 := CONCAT(_Nh_ADR_ROT,'/CFG/FRM/_', USINT_TO_STRINGF(aCfg[xR^.h.cf.c].frm,'%03d'),'.RW',USINT_TO_STRING(xL^.dsh));
//   _NhSdcVar(src := PTR_TO_UDINT(ADR( xR^.o.ob[0] )), siz := SIZEOF(NH_ROW_O)  );

//   _NhFrmName(read:=true, src:=ADR(xR^.o.ob[0]), cfg := aCfg[xR^.h.cf.c].frm, dsh:= xL^.dsh);

	rb:=_Nh_FRM_Read(frm:=USINT_TO_UINT(aCfg[xR^.h.cf.c].fBr), row := row);
   CASE xL^.dsh OF
     2:  //xR^.o    :=  _eRowBrw4;                                                 // dash ikony velke 3 riadkoy x 2 stlpce
         xIxB^.row.rws := 6;
         xIxB^.row.clm := 2;
         IF MOD(row,2) = 0 THEN
            x := xc + 5;
         ELSE
            x  := 0;
         END_IF;
         IF    row = 0 THEN y := 0;
         ELSIF row < 3 THEN y := y1 ;
         ELSIF row < 5 THEN y := y1 + xR^.o.ob[0].h      + 14;
         ELSIF row < 7 THEN y := y1 + xR^.o.ob[0].h * 2  + 28;
         ELSIF row < 9 THEN y := y1 + xR^.o.ob[0].h * 3  + 42;
         ELSIF row < 11 THEN  y := y1 + xR^.o.ob[0].h * 4  + 56;
         ELSE               y := y1 + xR^.o.ob[0].h * 5  + 70;
         END_IF;
         CASE xR^.h.cf.c OF
           1 : ;
           2 : ;
           3 : ;
           4 : ;
           5 : ;
          42 : ;
         ELSE
            IF xR^.o.ob[4].wh > 0 THEN                                           // ak je setup a nie je rom,cat,zon
               xR^.o.ob[4].x := xR^.o.ob[1].x +60;                               // pri malom DSH vypne stavovy obrazok
               xR^.o.ob[4].y := xR^.o.ob[1].y ;                                  // pri malom DSH vypne stavovy obrazok
            END_IF;
         END_CASE;

     3:  //xR^.o    :=  _eRowBrw12;                                                 // dash ikony male 12 riadkov x 2 stlpce
         IF yk > 1.0 THEN
            xIxB^.row.rws :=14;
//            xIxB^.row.rws :=12;
         ELSE
            xIxB^.row.rws :=12;
         END_IF;
         xIxB^.row.clm := 2;
         IF MOD(row,2) = 0 THEN
            x := xc;
         ELSE
            x  := 0;
         END_IF;
         IF    row = 0 THEN y := 0;
         ELSIF row < 3 THEN y := y1 ;
         ELSIF row < 5 THEN y := y1 + xR^.o.ob[0].h      + 10;
         ELSIF row < 7 THEN y := y1 + xR^.o.ob[0].h * 2  + 20;
         ELSIF row < 9 THEN y := y1 + xR^.o.ob[0].h * 3  + 30;
         ELSIF row <11 THEN y := y1 + xR^.o.ob[0].h * 4  + 40;
         ELSIF row <13 THEN y := y1 + xR^.o.ob[0].h * 5  + 50;
         ELSE               y := y1 + xR^.o.ob[0].h * 6  + 60;
         END_IF;
         IF aCfg[xR^.h.cf.c].fBr = 0 THEN
            xR^.o.ob[4].wh := 0;                                                 // pri malom DSH vypne stavovy obrazok
         END_IF;

   ELSE  //xR^.o          :=  _eRowBrw6;       // 1 siroky riadok = default, 1 stlpec
         IF yk > 1.0 THEN
            xIxB^.row.rws  := 7;
         ELSE
            xIxB^.row.rws  := 6;
         END_IF;
         xIxB^.row.clm  := 1;
         x              := 0;
         y              := (y1-5) + (xR^.o.ob[0].h+7) * USINT_TO_INT(row-1);

   END_CASE;
END_FUNCTION

FUNCTION _Nh_Row_BRW_Data {HIDDEN} : BOOL           //   NAPLNI RIADOK FIXNYMI HODNOTAMI
   VAR_INPUT
      //ref      : BOOL;
      row      : USINT;
      x        : USINT;
   END_VAR
   VAR_TEMP
      sld      : BOOL;
      blk      : BOOL;
//      cp       : USINT;
//      np       : INT;
      FgC      : USINT := 4;        // biela gulicka
      BgC      : USINT := 5;        // zlty slider
//      c        : USINT;
   END_VAR
   _Nh_Row_BRW_Data := true;
  _NhRowDSH(row := row);
   ii                := xR^.h.cf.c;
   aWeb.M[1].brw.r[0] :=  xR^;   aWeb.M[1].brw.r[0].o.ob[10].fmt := CONCAT(USINT_TO_STRING(ii),',',USINT_TO_STRING(row));
   xL^.brw            := true;
	_NhTypObr(cf:=xR^.h.cf.c, typ:=xDev^.cf.typ);
	xR^.o.ob[ 1].fn 	 := xObrWht^.obr;

   xR^.o.ob[ 1].cf    := xR^.h.cf;
   xR^.o.ob[ 2].cf    := xR^.h.cf;
   xR^.o.ob[ 4].cf    := xR^.h.cf;

   xR^.o.ob[ 9].cf.c  := 1;                                                   // nazov miestnosti
   xR^.o.ob[ 9].cf.n  := USINT_TO_INT(xDev^.cf.rom);                             // cislo

   xR^.o.ob[10].cf.c  := xR^.h.cf.c;                                          // nazov Dev
   xR^.o.ob[10].cf.n  := xR^.h.cf.n;                                          // nazov Dev
   sld                := aCfg[ii].sld;

   xO := ADR(xR^.o.ob[2]);                                                 // nampuje stavovy objekt [2]

   _Nh_Chk_FAV();

   CASE xR^.h.cf.c OF
(*
     6:  // HET
         xHet  := xDev;
         IF xR^.h.chk THEN

            pHet  := xPar;
            xPva  := ADR(pHet^.pva);
         ELSE
            xPva  := ADR(xHet^.me.pva);
         END_IF;
         _NhSetObjBrw(wh:=219,ob:=2, y:=xR^.o.ob[2].y-10,  h:= 33,  vb := adr(xHet^.me.tmp[100]), Fgc:=4, BgC:=1, o1 := 0, nTch:=1);                  // teplota HET
         _NhSetObjBrw(wh:=222,ob:=5,  vb := xPva);                                                    // predvolby 0,1,23 + zidana telota
         IF xL^.dsh > 1 THEN
            xR^.o.ob[5].x  := xR^.o.ob[3].x;                            // hand/auto dat na poziciu oblubene
            xR^.o.ob[3].wh := 0;                                        // oblubene nebude
            xR^.o.ob[4].wh := 0;                                        // setup nebude
         END_IF;
         IF xL^.dsh < 3 THEN
            IF xHet^.me.own[99] THEN
               _NhSetObjBrw(ob:=7, wh:=219, x:=xR^.o.ob[2].x-5, y:=xR^.o.ob[2].y+35 ,  h:= 22,  vb := adr(xHet^.me.tmp[99]), Fgc:=16, BgC:=1, o1 := 0, nTch:=1);                  // teplota HET
            END_IF;
         ELSE
            xR^.o.ob[2].y := xR^.o.ob[10].y;                         // teplotu vratit na uroven nazvu
            xR^.o.ob[2].w := 25;                                     // teplotu vratit na uroven nazvu
            xR^.o.ob[10].cf.p := 6;                                  // 8 - znakov nazvu
         END_IF;
         xR^.o.ob[1].wh := 9;
         xR^.o.ob[1].fn := 0;
*)
    10: // SVD
         _NhSetObjBrw(wh:=7,ob:=7, w:=48, cm := 44,  vb := ADR(vr));        // zobrazenie blokovania PIR nad stavovym obrazkom
          xR^.o.ob[ 2].wh := 9;
    11:   _NhSetObjBrw(wh:=7,ob:=7, w:=48, cm := 44, vb := ADR(vr));        // zobrazenie blokovania PIR nad stavovym obrazkom  // SVA
          xR^.o.ob[ 2].wh := 9;
    12:   // RGB
          _NhSetObjBrw(wh:=7,ob:=7, w:=48, cm := 44, vb := ADR(vr));        // zobrazenie blokovania PIR nad stavovym obrazkom
          xR^.o.ob[ 2].wh := 9;
    13:  // WSB
         _NhSetWSB(o := 1, chk := xR^.h.chk);
//         _NhSetObjBrw(ob := 5, sl := 1, o1  := 127, o2 := 129, vb := ADR(xDev^.ok.blk));
    14:  // TLA
         _NhSetWSB(o := 1, chk := xR^.h.chk);

(*
    23:  // VEN
//         xR^.o.ob[ 6].wh := 7;   // cas do vypnutia / PIR, blokovanie
         _NhSetObjBrw(wh:=7,ob:=7, w:=48, cm := 44, vb := ADR(vr));        // zobrazenie blokovania PIR nad stavovym obrazkom
         xVen := xDev;
         IF xVen^.cf.typ < 1 THEN
            sld := 0;
         END_IF;
*)

    35:  // BLK
         xR^.o.ob[ 2].wh   := 9;
    36:  // TIM
         xR^.o.ob[ 2].wh   := 9;
    37:  // BRA
         _NhSetObjDsh(grp := 37);
//         sld   := false;                                                // nasilne sa zrusi slider

    40:  // TGL

          _NhSetWSB(o := 1, chk := xR^.h.chk);
    42:  ;// DLM
(*
         xDLm  := xDev;
         xPtD  := ADR(xR^.o.ob[9].cf.n);
         xPtD^ := PTR_TO_UDINT( ADR(xDlm^.hw.txt) );
*)

    43:  ;// DLS
         sld   := false;
//         xDLs  := xDev;
//         _NhSetObjBrw(wh := 251, ob := 5, sl := USINT_TO_SINT(row), vb := ADR(xDLs^.hw.set.ActualLevel));

    44:  ;// DLQ

   ELSE

   END_CASE;

   CASE xR^.h.cf.c OF
     4:  // SCN
         xO^.wh := 3;
         xR^.o.ob[ 6].wh := 7;   // SVD
     5:  // ACT

     7:  // KOT

//         _NhSetObjBrw(wh := 222, ob:=5, vb := ADR(vr));
//         sld := 0;

//         xR^.o.ob[ 9].wh := 0;                      // nevypisuje sa druhy riadok
//         _NhSetObjBrw(wh := 222, ob := 5, w := 48, h := 68, c:= 3, n := 1, vb := ADR(xHet^.cx.ter));

     8:  // TVE

     9:  // CER
//         _NhSetObjBrw(wh := 222, ob:=5, vb := ADR(vr));
//         sld := 0;

//         xR^.o.ob[ 9].wh := 0;                      // nevypisuje sa druhy riadok
//         _NhSetObjBrw(wh := 222, ob := 5, w := 48, h := 68, c:= 3, n := 0, vb := ADR(xCfx^));

    15:  // PIR
         blk               := xR^.h.chk = false;                                       // blk len ked nie je vo vazbe
         IF xR^.h.chk THEN
            _NhxDev2(c := xR^.o.ob[ 4].cf.c, n := xR^.o.ob[ 4].cf.n, x:=13);
            IF xDev2^.cf.rom = 0 THEN
               _NhxDev2(c := xR^.h.cf.c , n := xR^.h.cf.n, x:=14);
            END_IF;
            _NhShwDay(cf := 1, nr := xDev2^.cf.rom, rom := false);
            xR^.o.ob[ 8].y   :=xR^.o.ob[ 8].y  + xR^.o.ob[ 1].w / 2;                      // pozicia DAY-mode bude dolu
//         ELSE
//            xR^.o.ob[ 2].wh   := 3;

         ELSIF xDev^.cf.typ = 1 THEN
            _NhSetObjBrw(wh:=200, ob := 6, w := 48, h:= 0, FgC := 8, c := 0, vb := ADR(xDev^.al.Off ), nTch:=1 );     // pritomnost tamperu na pir
         END_IF;

    16:  // TER
         _NhSetObjBrw(ob:=2, wh:=219, vb := adr(xDev^.al.ou.val),BgC:=1);
         blk := true;
    17:  // TER
         _NhSetObjBrw(ob:=2, wh:=219, vb := adr(xDev^.al.ou.val),BgC:=1);
         blk := true;
    18:  // TER
         _NhSetObjBrw(ob:=2, wh:=219, vb := adr(xDev^.al.ou.val),BgC:=1);
         blk := true;

    19:  // LUX
         _NhSetObjBrw(ob:=2, wh:=219, vb := adr(xDev^.al.ou.val),BgC:=1,fmt := '%4.0f%%');
         blk := true;
//         _NhSetObjBrw(vb := ADR(xDev^.al.ou.val),  wh := 255, ob := 2);

    20:  // FAV LIST
         xO^.wh   := 1 ;                               // len obrazok
         xO^.cm   := 27 ;                             // zmena oblubeneho
         xFav     := xDev;
         IF xFav^.cx = xA^.fav THEN
            xR^.o.ob[ 2].fn := 38;
         ELSE
            xR^.o.ob[ 2].fn := 35;
         END_IF;
         xR^.o.ob[ 3].wh := 0;
         xR^.o.ob[ 4].wh := 0;
         IF xFav^.cx.n > 0 THEN
            xR^.o.ob[ 9].cf.c := 22; xR^.o.ob[ 9].cf.n := USINT_TO_INT(xFav^.cx.c);      // do 2.riadku cislo usra
         ELSE
            xR^.o.ob[ 9].wh := 0;                      // nevypisuje sa druhy riadok
         END_IF;

    21:  xR^.o.ob[ 6].wh := 7;   // ZAS

    22:  xR^.o.ob[ 1].cm := 201;   // USR - WEB_FRM
         xR^.o.ob[ 4].wh := 0;                         // nebude text 2
         xR^.o.ob[ 9].wh := 0;                         // nebude text 2
         xR^.o.ob[ 2].wh := 1;                           // vypisat check
//         xR^.o.ob[ 2].fn := 35;
         xR^.o.ob[ 2].w  := 72;                       // vypisat check

    24:  // KEY;
         xR^.o.ob[ 4].cm := 81;                         // zatial posde do ROM

    33:
    38:  // RFI
         xRFI := xDev;
         _NhSetObjBrw(ob := 5, sl := 1, o1  := 127, o2 := 129, vb := ADR(xRFI^.cx.blk));

         _NhSetObjBrw(ob := 6, sl := 2, o1  := 275, o2 := 276, vb := ADR(xRFI^.cx.Beep), w:= 48 );
         _NhSetObjBrw(ob := 7, sl := 3, o1  := 270, o2 := 271, vb := ADR(xRFI^.cx.LedG), w:= 32 );
         _NhSetObjBrw(ob := 8, sl := 4, o1  := 270, o2 := 272, vb := ADR(xRFI^.cx.LedR), w:= 32 );

    39:  // RFK
         IF xM^.new = xR^.h.nd THEN                // novo pridany alebo najdena karta zmeni farbu boxu na zeleno
            xM^.new := 0;
            xR^.o.ob[0].FgC   := 8;
            xR^.o.ob[0].BgC   := 1;
         END_IF;

   ELSE  ;
//      _NhSetObjBrw(wh := xR^.h.cf.c, ob := 2, vb := ADR(xR^.o.ob[2].cf.n) );
   END_CASE;
   IF sld  THEN                                         // nadefinuje slider
      rb := _NhSetObjBrw(wh := 250, ob := 5, sl := USINT_TO_SINT(row), vb := ADR(xDev^.al.in.val), t:= 0, w:=_Nh_O12(xL^.dsh<2,350,160), FgC := Fgc,BgC := BgC,  x:= xR^.o.ob[5].x );
      IF xL^.dsh > 2 THEN
         xR^.o.ob[2].wh := 0;                            // pri malom DSH vypne stavovy obrazok
         xR^.o.ob[6].wh := 0;                            //
      END_IF;
   ELSIF blk   THEN
      _NhSetObjBrw(wh:=200, ob := 5, w := 48, h:= 0, FgC := 4, c := 0, vb := ADR(xDev^.cf.blk ) );     // blokovat (ON/OFF)
   END_IF;

(*
   IF xL^.dsh > 2 THEN                                      // pri malom DSH sa posunie hodnota dolu
      IF xR^.o.ob[2].wh = 19 AND xR^.o.ob[2].fn = 0 THEN    // len hodnota bez podkladu BTN
         xR^.o.ob[2].y   := xR^.o.ob[2].y+60;
      END_IF;
   END_IF;
*)

END_FUNCTION

FUNCTION _NhBrwND {HIDDEN} : BOOL         // vrati index odpovedajuci cf
   VAR_INPUT
      rws      : SINT := 11;
   END_VAR
   _NhBrwND := 1;
   WHILE nd > 2 AND rws > 0 DO
      nd := nd - 1 ;
      IF _NhxDev(c := cf, n := nd, x:=252 ) THEN
         rws := rws - 1;
      END_IF;
   END_WHILE;
END_FUNCTION

FUNCTION _NhBrwIX {HIDDEN} : INT         // vrati index odpovedajuci cf
   VAR_INPUT
      cf    : USINT;
   END_VAR
   _NhBrwIX := 1;
   WHILE _Nh_IxC[_NhBrwIX] > 0 AND _Nh_IxC[_NhBrwIX] <> cf DO
      _NhBrwIX := _NhBrwIX + 1;
   END_WHILE;
END_FUNCTION

VAR_GLOBAL
   row      {HIDDEN} : USINT;
   nx       {HIDDEN} : USINT;
END_VAR

FUNCTION  _Nh_Web_BRW {HIDDEN} : BOOL     // RIADKOVY BROWSER
   VAR_TEMP
      brw      :  BOOL := true;        // z indexu prenesie data do row browseru
      wht      :  USINT;
   END_VAR
   VAR_TEMP
      row0     : BOOL;
      kx       : INT;
//      ya       : INT;
   END_VAR
   _Nh_Web_BRW   := true;
//   aSys.cnt    := aSys.cnt + 1;
   xIxB := ADR(xM^.ixb[0]);
   IF xIxB^.idx = 0 OR xM^.wht >= 20 THEN                                                   // novy index, vypis od prvej vety
      _Nh_Brw_Idx();                                                                           // vymaze vsetko a vytvori novy index

   END_IF;

   GC_Begin(GrData := xCan);
   GC_ReSetOrigin(GrData := xCan);
   CASE xM^.wht OF
     -1: // len refresh riadkov
         brw := false;
     -2: // refresh   Frame (len menu)
         brw := false;
      1: // dolu
         IF xM^.iter = 0 THEN
            xM^.iter    := 1;                                                    // krd sa sem vrati v druhom cykle uz sem nepojde
            brw         := false;                                                // len sa prekresli co je na obrazovke, nie nove data
            xA^.tch.cmd := 255;                                                  // v druhom cykle ide rovno sem
            _Nh_Web_BRW   := false;                                                // zabezpeci, aby sa neresetol cmd
            IF xIxB^.ix1 > 1 THEN
               row0        := true;                                              // vykresli sa riadok, aj sa skoriguje suradnica y
               IF xL^.dsh = 1 THEN
                  GC_MoveTo(x:=0,y:= 95,GrData := xCan);                               // posun dolu
//                  GC_MoveTo(x:=0,y:= 95,GrData := xCan);                               // posun dolu
               ELSE
                  GC_MoveTo(x:=0,y:= 0,GrData := xCan);                               // posun dolu
                  row0        := false;                                              // vykresli sa riadok, aj sa skoriguje suradnica y
               END_IF;
               xM^.delay   := 1;                                                 // vylistuje sa prazna cast riadka a caka sa, aby sa vratila obrazovka
            ELSE                                                                 // nie je dalsi riadok
               GC_MoveTo(x:=0,y:= 45,GrData := xCan);                               // posun dolu
               xM^.delay := 500;                                                 // vylistuje sa prazna cast riadka a caka sa, aby sa vratila obrazovka
              END_IF;
            GC_SetOrigin(GrData := xCan);                                        // prestavi na tendo cyklus

         ELSE
            _NhSet1Row(fnd := false, dn := true, row := xIxB^.row.rws );
            xM^.iter := 0;                                                       // vrati sa do povodnehostavu
         END_IF;

      2: // hore
         IF xM^.iter = 0 THEN
            xM^.iter    := 1;                                                    // krd sa sem vrati v druhom cykle uz sem nepojde
            brw         := false;                                                // len sa prekresli co je na obrazovke, nie nove data
            xA^.tch.cmd := 255;                                                  // v druhom cykle ide rovno sem
            _Nh_Web_BRW   := false;                                                // zabezpeci, aby sa neresetol cmd
            IF xIxB^.ix2 < xIxB^.idx AND xB^.rw > 0 THEN
               row0        := true;                                              // vykresli sa riadok, aj sa skoriguje suradnica y
               IF xL^.dsh = 1 THEN
                  GC_MoveTo(x:=0,y:=-50,GrData := xCan);                               // posun hore
//                  GC_MoveTo(x:=0,y:=-90,GrData := xCan);                               // posun hore
               ELSE
                  GC_MoveTo(x:=0,y:=0,GrData := xCan);                               // posun hore
                  row0        := false;                                              // vykresli sa riadok, aj sa skoriguje suradnica y
               END_IF;
               xM^.delay   := 1;                                                 // vylistuje sa prazna cast riadka a caka sa, aby sa vratila obrazovka
            ELSE                                                                 // nie je dalsi riadok
               xM^.delay := 500;                                                 // vylistuje sa prazna cast riadka a caka sa, aby sa vratila obrazovka
               GC_MoveTo(x:=0,y:=-45,GrData := xCan);                               // posun hore
            END_IF;
             GC_SetOrigin(GrData := xCan);                                        // prestavi na tendo cyklus
         ELSE
            _NhSet1Row(fnd := false, up := true, row := xIxB^.row.rws );         // ziskaju sa nove data od 1.riadka
            xM^.iter := 0;                                                       // vrati sa do povodneho stavu
         END_IF;

     10: // vypis od 1.riadka s predefinovanim dat v riadku, nie novy index
         _Nh_Map_Idx(ixb := 0, idx := xIxB^.ix1);

     15 : // zmazat vetu = novy index a refresh od 1.riadku alebo za DEL-rec
         _NhSet1Row(fnd := false, del := true);                                     // nastavi rw1 no-del vetu
         _Nh_Brw_Idx();                                                             // vytvori novy index bez zmazaneho zaznamu
         wht := 25;                                                                 // vypis od zapamatanej vety

     20: // vytvoreny novy index, refresh tak aby zapamatana veta zostala v 1.riadku
         xIxB^.ix1 := 1;
         _NhSet1Row(fnd := false);                                     // nastavi rw1 no-del vetu
//         _NhSet1Row(fnd := false);

     25: // navrat spat = vytvorit novy index, vypis od zapamatanej vety v 1.RIADKU
          wht    := 25;

     30 : // nova veta   = novy index a pridanu vetu zobrazit na konci browsu ak sa da
            _NhSet1Row(end := true);
   END_CASE;
   CASE wht OF
     25 :   // najde v indexe vetu, ktora odpoveda zapamatanej vete a to bude 1.veta v browse = posunie vetu na 1.riadok
            _NhSet1Row();
   END_CASE;

   row   := 1; //xIxB^.ix1;
   nx    := xIxB^.ix1;                                      // index na data
   // xIdx je namapovane na vetu xIxB^.ix1;
   // xIxB je namapovane na sadu dat pre browser xM^.ixb[0]
   xB^.rw  := 0;

//IF false THEN

   IF xL^.obj > 200 THEN
      WHILE nx > 0 AND row <= xIxB^.row.rws DO
         xR := ADR(xB^.r[ row  ]);
         IF nx <= xIxB^.idx THEN                                        // mame vetu
            xB^.rw      := row;                                             // posledny naplneny ridok
            xIxB^.ix2   := nx;
            IF xL^.obj=255 THEN
					yTx2	:= CONCAT('Err:_Nh_Web_BRW,xL^.obj=255: nx:',USINT_TO_STRING(nx),' row:',USINT_TO_STRING(row),' c:',USINT_TO_STRING(xR^.h.cf.c),' n:',INT_TO_STRING(xR^.h.cf.n))  ;
   	 			rb		:= _Nh1RowTxt(logRst := 1);
					aSys.ErrPt	:= aSys.ErrPt + 1;
(*
               nx             := nx + 1;
               xR^.o.ob[0]    := _eRowBrw6.ob[0];       // 1 siroky riadok = default, 1 stlpec
               xR^.o.ob[1]    := _eRowBrw6.ob[1];       // 1 siroky riadok = default, 1 stlpec
               xR^.o.ob[1].wh := 255;
               xR^.h.cf       := xIdx^.ix[aWeb.nbr].dev;
               x              := 0;
               y              := (y1-5) + (xR^.o.ob[0].h+7) * USINT_TO_INT(row-1);
               _Nh_Shw_Obj(row:=row,x := x, y:= y);                         // koriguje x,y o kazdeho objektu riadka a vykresli
*)
            END_IF;
         END_IF;
         xIdx  := xIdx + SIZEOF(NH_IDX);
         row   := row + 1;
      END_WHILE;
   ELSE
      WHILE nx > 0 AND row <= xIxB^.row.rws DO
         xR := ADR(xB^.r[ row  ]);
         yIdxR       := xIdx^.ix[aWeb.nbr];                                   // nove od 21.10.22
         IF brw THEN                                     						// natahuju sa struktiry kazdej vety nanovo
            IF nx <= xIxB^.idx THEN                                        // mame vetu
               kx := 0;
               xR^.h.cf    := xIdx^.ix[aWeb.nbr].dev;
					IF xR^.h.cf.c > 0 THEN
						IF yIdxR.chk AND yIdxR.vaz AND yIdxR.nd > 0 THEN
	                  xR^.h.nd    := yIdxR.nd;
						ELSE
	                  xR^.h.nd    := USINT_TO_INT(nx);
   					END_IF;
                  xIxB^.ix2   := nx;
                  nx          := nx + 1;

                  _NhxCfg(c := xR^.h.cf.c, n := xR^.h.cf.n, par := true, p := xR^.h.cf.p, x:=19);                     // xDev,xCfg,xPar pre aktualny riadok
                  IF aCfg[xR^.h.cf.c].fBr > 0 THEN
                     _Nh_Frm_Row_BRW(row := row, new := true);
                  ELSE
                     _Nh_Row_BRW_Data(row := row , x:=11);                                                              // naplni riadky
                  END_IF;

                  IF xM^.new = USINT_TO_INT(row) THEN                		// je DEL, alebo CPY - dodefinuje objekt namiesto obj[1]
                     IF xA^.tch.del OR xA^.tch.cpy THEN
                    		_NhSetObjBrw( wh := 202, vb := adr(vr) );
                       	x           := x -94;
							ELSE
	                     xM^.new := 0;
                     END_IF;
                  END_IF;
               ELSE
                  yTx2     := CONCAT('ERR!-02 _NhWebBrw vypis idx/nx/c/n: ',
                           USINT_TO_STRING(xIxB^.idx),'/',USINT_TO_STRING(nx),'/',USINT_TO_STRING(xR^.h.cf.c),'/',INT_TO_STRING(xR^.h.cf.n));
                  _Nh1RowTxt(logRst := 1, adTime := 3);
                  EXIT;
               END_IF;
            ELSE
               EXIT;
            END_IF;
         ELSE
            x  := 0;
            y  := 0;
         END_IF;
         IF xR^.h.nd > 0 AND xR^.h.cf.c > 0 THEN
             xB^.rw  := row;                                             // posledny naplneny ridok
            _NhxCfg(c := xR^.h.cf.c, n := xR^.h.cf.n, par := true, p := xR^.h.cf.p, x:=19);                     // xDev,xCfg,xPar pre aktualny riadok
            IF aCfg[xR^.h.cf.c].fBr > 0 THEN
               _Nh_Frm_Row_BRW(row := row);
            END_IF;
//  				_Nh_Shw_Obj(row:=row, x := x, y:= y);                         // koriguje x,y o kazdeho objektu riadka a vykresli

				IF xR^.h.new THEN
    				_Nh_Shw_Obj(row:=row);                         				// koriguje x,y o kazdeho objektu riadka a vykresli
				ELSE
    				_Nh_Shw_Obj(row:=row, x := x, y:= y);                    // koriguje x,y o kazdeho objektu riadka a vykresli
//					IF xM^.wht = -1 AND xR^.h.cf.c = 31 THEN     				// vynimka pre rolety
//					IF xR^.h.cf.c = 31 THEN     										// vynimka pre rolety
//						xR^.h.new := true;
//					END_IF;
				END_IF;
         ELSE
            EXIT;
         END_IF;
         xIdx  := xIdx + SIZEOF(NH_IDX);
         row   := row + 1;
      END_WHILE;

(*
//   IF row0 THEN                                                      // dodatocny vypis riadka 0/7 pri rorovani hore dolu
   IF false THEN                                                      // dodatocny vypis riadka 0/7 pri rorovani hore dolu
      IF xM^.wht = 2 THEN
         row := 7;
//**-**         _NhMapIdx(ixb := 0, idx := xIxB^.ix1, idx := xIxB^.ix2 + 1);
         _Nh_Map_Idx(ixb := 0, idx := xIxB^.ix2 + 1);
         xB^.xy.yp := 0;
      ELSE
         row := 1;
//**-**         _NhMapIdx(ixb := 0, idx := xIxB^.ix1, idx := xIxB^.ix1 - 1);
         _Nh_Map_Idx(ixb := 0, idx := xIxB^.ix1 - 1);
         xB^.xy.yp := -kyr;
      END_IF;

         xR 			:= ADR(xB^.r[ 0  ]);
         xR^.h.cf    := xIdx^.ix[aWeb.nbr].dev;
         xR^.h.nd    := USINT_TO_INT(xIxB^.ix2+1);

         IF xR^.h.cf.c > 0 THEN
            _NhxCfg(c := xR^.h.cf.c, n := xR^.h.cf.n, par := true, n := xR^.h.cf.p, x:=20);                     // xDev,xCfg,xPar pre aktualny riadok
            IF aCfg[xR^.h.cf.c].fBr > 0 THEN
               _Nh_Frm_Row_BRW(row := row, new := true);
            ELSE
               _Nh_Row_BRW_Data(row := row , x:=12);                                                              // naplni riadky
            END_IF;
            _Nh_Shw_Obj(row:=0, y := y + xB^.xy.yp);                         // koriguje x,y o kazdeho objektu riadka a vykresli
         END_IF;

      END_IF;
*)

   END_IF;
//END_IF;

   GC_ReSetOrigin(GrData := xCan);
   _NhShwMnu();
   _NhPgNav();

   GC_End(GrData := xCan);
END_FUNCTION

{ $ END_IF }
